FUNCTION_BLOCK E_DELAY
  (* Version 1.0, 2005-05-17, Goran Cengic, Chalmers *)
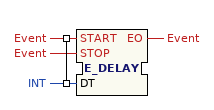
  EVENT_INPUT
    START WITH DT;
    STOP;
  END_EVENT
  EVENT_OUTPUT
    EO;
  END_EVENT
  VAR_INPUT
    DT : INT;
  END_VAR
END_FUNCTION_BLOCK
